{attribute 'qualified_only'}
{attribute 'strict'}
TYPE E_TakeMode :
(
	None := 0,// 不动作
	Take0,// 取Line0料
	Take1,// 取Line1料
	Take3Load,// 取Line3上料站 产品
	Place1,// 放Line1料
	Place3Load// 放线体3上料站
);
END_TYPE

(* stored: Version 1.1.0.1, ProductVersion 3.1.4024.3
   DUT E_TakeMode: Id {3bb012a5-b6ca-4f7e-8633-c1cefe630a23} *)
